PROGRAM MAIN
VAR
	fbOperate : FB_Operate;
END_VAR

F_UpdateIO();

fbOperate(iq_eOperation := GVL_Operation.iq_eOperation,
	iq_eTransportTube := GVL_Operation.iq_eTransportTube,
	i_bCancel := GVL_Operation.i_bCancel,
	q_bBusy => GVL_Operation.q_bBusy);
	
GVL_Operation.i_bCancel := FALSE; // Acknowledge the cancel flag

END_PROGRAM

(* stored: Version 1.1.0.1, ProductVersion 3.1.4024.0
   POU MAIN: Id {e39c3acf-17bf-44fe-a884-c77329dee9c5}, SpecialFunc None *)
